PROGRAM Main
VAR
    // Motors
    // MRCO Axes
    {attribute 'TcLinkTo' := '.bLimitForwardEnable:=TIIB[GasNozzleX-EL7047]^STM Status^Status^Digital input 2;
                              .bLimitBackwardEnable:=TIIB[GasNozzleX-EL7047]^STM Status^Status^Digital input 1'}
    {attribute 'pytmc' := '
        pv: TMO:MRCO:MMS:01
    '}
    M1 : DUT_MotionStage := (bPowerSelf:=TRUE,
    nEnableMode:=ENUM_StageEnableMode.ALWAYS,
    nBrakeMode:= ENUM_StageBrakeMode.NO_BRAKE ); // Gas Nozzle X

    {attribute 'TcLinkTo' := '.bLimitForwardEnable:=TIIB[GasNozzleY-EL7047]^STM Status^Status^Digital input 2;
                              .bLimitBackwardEnable:=TIIB[GasNozzleY-EL7047]^STM Status^Status^Digital input 1'}
    {attribute 'pytmc' := '
        pv: TMO:MRCO:MMS:02
    '}
    M2 : DUT_MotionStage := (bPowerSelf:=TRUE,
    nEnableMode:=ENUM_StageEnableMode.ALWAYS,
    nBrakeMode:= ENUM_StageBrakeMode.NO_BRAKE); // Gas Nozzle Y

    {attribute 'TcLinkTo' := '.bLimitForwardEnable:=TIIB[GasNozzleZ-EL7047]^STM Status^Status^Digital input 1;
                              .bLimitBackwardEnable:=TIIB[GasNozzleZ-EL7047]^STM Status^Status^Digital input 2'}
    {attribute 'pytmc' := '
        pv: TMO:MRCO:MMS:03
    '}
    M3 : DUT_MotionStage := (bPowerSelf:=TRUE,
    nEnableMode:=ENUM_StageEnableMode.ALWAYS,
    nBrakeMode:= ENUM_StageBrakeMode.NO_BRAKE); // Gas Nozzle Z

    {attribute 'TcLinkTo' := '.bLimitForwardEnable:=TIIB[SamplePaddleX-EL7047]^STM Status^Status^Digital input 2;
                              .bLimitBackwardEnable:=TIIB[SamplePaddleX-EL7047]^STM Status^Status^Digital input 1'}
    {attribute 'pytmc' := '
        pv: TMO:MRCO:MMS:04
    '}
    M4 : DUT_MotionStage := (bPowerSelf:=TRUE,
    nEnableMode:=ENUM_StageEnableMode.ALWAYS,
    nBrakeMode:= ENUM_StageBrakeMode.NO_BRAKE); // Sample Paddle X

    {attribute 'TcLinkTo' := '.bLimitForwardEnable:=TIIB[SamplePaddleY-EL7047]^STM Status^Status^Digital input 2;
                              .bLimitBackwardEnable:=TIIB[SamplePaddleY-EL7047]^STM Status^Status^Digital input 1'}
    {attribute 'pytmc' := '
        pv: TMO:MRCO:MMS:05
    '}
    M5 : DUT_MotionStage := (bPowerSelf:=TRUE, 
    nEnableMode:=ENUM_StageEnableMode.ALWAYS,
    nBrakeMode:= ENUM_StageBrakeMode.NO_BRAKE); // Sample Paddle Y

    {attribute 'TcLinkTo' := '.bLimitForwardEnable:=TIIB[SamplePaddleZ-EL7047]^STM Status^Status^Digital input 2;
                              .bLimitBackwardEnable:=TIIB[SamplePaddleZ-EL7047]^STM Status^Status^Digital input 1'}
    {attribute 'pytmc' := '
        pv: TMO:MRCO:MMS:06
    '}
    M6 : DUT_MotionStage := (bPowerSelf:=TRUE,
    nEnableMode:=ENUM_StageEnableMode.ALWAYS,
    nBrakeMode:= ENUM_StageBrakeMode.NO_BRAKE); // Sample Paddle Z

    // MRCO Axes
    fbMotionStageM1 : FB_MotionStage;
    fbMotionStageM2 : FB_MotionStage;
    fbMotionStageM3 : FB_MotionStage;
    fbMotionStageM4 : FB_MotionStage;
    fbMotionStageM5 : FB_MotionStage;
    fbMotionStageM6 : FB_MotionStage;  
END_VAR

// Hardware Enable
//Mrco
// Gas Nozzle
M1.bHardwareEnable := TRUE;
M2.bHardwareEnable := TRUE;
M3.bHardwareEnable := TRUE;
// Sample Paddle
M4.bHardwareEnable := TRUE;
M5.bHardwareEnable := TRUE;
M6.bHardwareEnable := TRUE;
    
// fbMotionStage
// MRCO
// Gas Nozzle
fbMotionStageM1(stMotionStage:=M1);
fbMotionStageM2(stMotionStage:=M2);
fbMotionStageM3(stMotionStage:=M3);
// Sample Paddle
fbMotionStageM4(stMotionStage:=M4);
fbMotionStageM5(stMotionStage:=M5);
fbMotionStageM6(stMotionStage:=M6);

END_PROGRAM

(* stored: Version 1.1.0.1, ProductVersion 3.1.4022.18
   POU Main: Id {3f08c9da-acd6-4059-bcf8-867945acb3ea}, SpecialFunc None *)
